Staubli VAL3: push.pgx

public program push(Queue& x_qQueue, MotionCmd& x_mCmd, bool& x_bRes)
begin
  // Copyright (c) 2016, Ocado Technology - Robotics Research Team
  //
  // Licensed under the Apache License, Version 2.0 (the "License");
  // you may not use this file except in compliance with the License.
  // You may obtain a copy of the License at
  //
  //     http://www.apache.org/licenses/LICENSE-2.0
  //
  // Unless required by applicable law or agreed to in writing, software
  // distributed under the License is distributed on an "AS IS" BASIS,
  // WITHOUT WARRANTIES OR CONDITIONS OF ANY KIND, either express or implied.
  // See the License for the specific language governing permissions and
  // limitations under the License.



  if (x_qQueue.nElems < size(x_qQueue.buffer))
    x_qQueue.buffer[x_qQueue.nPush] = x_mCmd
    x_qQueue.nElems = x_qQueue.nElems + 1
    x_qQueue.nPush = x_qQueue.nPush + 1
    if (x_qQueue.nPush >= size(x_qQueue.buffer))
      x_qQueue.nPush = 0
    endIf
    x_bRes = true
  else
    x_bRes = false
  endIf
end
